FUNCTION_BLOCK FB_MockCylinder IMPLEMENTS I_Cylinder
VAR
    _Extended  : BOOL;
    _Retracted : BOOL := TRUE;
    
    ExtendCallCount  : INT := 0;
    RetractCallCount : INT := 0;
END_VAR

METHOD Extend
_Extended := TRUE; 
_Retracted := FALSE; 
ExtendCallCount := ExtendCallCount + 1;
END_METHOD

PROPERTY Extended : BOOL
GET
Extended := _Extended;
END_GET
END_PROPERTY

METHOD Retract
_Extended := FALSE; 
_Retracted := TRUE; 
RetractCallCount := RetractCallCount + 1;
END_METHOD

PROPERTY Retracted : BOOL
GET
Retracted := _Retracted;
END_GET
END_PROPERTY

END_FUNCTION_BLOCK

(* stored: Version 1.1.0.1, ProductVersion 3.1.4024.15
   POU FB_MockCylinder: Id {f01286c1-7ad8-4665-be6d-b1d10066815f}, SpecialFunc None
   Method Extend: Id {98721f0e-fbdf-498b-aff3-c02e8b40e405}
   Property Extended: Id {9f1d5f9b-9529-4cf8-a7f5-73c380daae19}
   Get Get: Id {10bdb286-10e9-4dac-9a5d-643bc99f0abd}
   Method Retract: Id {c0a20e65-920a-4182-9765-19b79d027175}
   Property Retracted: Id {791cb054-55f7-4508-83e6-e7878573b647}
   Get Get: Id {dac08ce4-8457-48b3-91ba-217cf6badbfd} *)
